{attribute 'linkalways'} 
{attribute 'no_explicit_call' := 'This FB is a CLASS and must be accessed using methods or properties'}
FUNCTION_BLOCK Feeder EXTENDS CyclicInstance IMPLEMENTS I_Feeder
VAR
	_nci : I_Nci;
	_fb : FB_NciFeedTable;
	_table : ST_NciFeedGroupTable;
	_execute : BOOL;
	_reset : BOOL;
	_feedDone : BOOL;
	_channelDone : BOOL;
	_feedBusy : BOOL;
	_resetBusy : BOOL;
	_error : BOOL;
	_errorId : UDINT;
	
	state : (IDLE, RESETTING, FEEDING, DONE, ERROR);
	command : (NONE, RESET, FEED);
	
	commandFeedback : I_CommandFeedbackReadWrite;
END_VAR

PROPERTY ChannelDone : BOOL
GET
ChannelDone := _fb.bChannelDone;
END_GET
END_PROPERTY

METHOD  CyclicCall
CASE state OF
	IDLE:
		_fb(
			bExecute := FALSE,
			bReset := FALSE,
			stNciToPlc := _nci._InternalNciPlcRef.nciToPlc,
			stFeedGroupTable := _table,
			bFeedingDone => _feedDone,
			bChannelDone => _channelDone,
			bFeedBusy => _feedBusy,
			bResetBusy => _resetBusy,
			bError => _error,
			nErrorId => _errorId
		);
		
		CASE command OF
			RESET:
				state := RESETTING;
				command := NONE;
				commandFeedback.SetBusy();
			FEED:
				state := FEEDING;
				command := NONE;
				commandFeedback.SetBusy();
		END_CASE

	RESETTING:
		_fb(
			bExecute := FALSE,
			bReset := TRUE,
			stNciToPlc := _nci._InternalNciPlcRef.nciToPlc,
			stFeedGroupTable := _table,
			bChannelDone => _channelDone,
			bFeedBusy => _feedBusy,
			bResetBusy => _resetBusy,
			bError => _error,
			nErrorId => _errorId
		);
		
		IF NOT _fb.bResetBusy THEN		
			IF _fb.bError THEN
				state := ERROR;
			ELSE
				state := DONE;
			END_IF
		END_IF

	FEEDING:
		_fb(
			bExecute := TRUE,
			bReset := FALSE,
			stNciToPlc := _nci._InternalNciPlcRef.nciToPlc,
			stFeedGroupTable := _table,
		);
		
		IF NOT _fb.bFeedBusy THEN
			IF _fb.bError THEN
				state := ERROR;
			ELSIF _fb.bFeedingDone THEN
				state := DONE;
			END_IF
		END_IF
	
	DONE:
		IF commandFeedback <> 0 THEN
			commandFeedback.SetDone();
		END_IF
		state := IDLE;		
	ERROR:
		IF commandFeedback <> 0 THEN
			commandFeedback.SetError(_fb.nErrorId);
		END_IF
		state := IDLE;
ELSE
	state := IDLE;
END_CASE
END_METHOD

METHOD FB_init : BOOL
VAR_INPUT
	bInitRetains : BOOL; // if TRUE, the retain variables are initialized (warm start / cold start)
	bInCopyCode : BOOL;  // if TRUE, the instance afterwards gets moved into the copy code (online change)
	nci : I_Nci;
END_VAR
IF nci <> 0 THEN
	_nci := nci;
END_IF
END_METHOD

METHOD FeedTable
VAR_INPUT
	table : I_Table;
	feedback : REFERENCE TO I_CommandFeedback;
END_VAR
VAR
	pCmd : POINTER TO FeederCommand;
END_VAR
IF NOT IsAlreadyExecuting() THEN
	_table := table._InternalTable;
	command := FEED;
	SetupFeedback(Feedback);
END_IF
END_METHOD

METHOD PRIVATE IsAlreadyExecuting : BOOL
IF commandFeedback = 0 THEN
	RETURN;
END_IF

IsAlreadyExecuting := commandFeedback.Busy;
END_METHOD

PROPERTY LogFeederEntries : BOOL
GET
LogFeederEntries := _fb.bLogFeederEntries;
END_GET
SET
_fb.bLogFeederEntries := LogFeederEntries;
END_SET
END_PROPERTY

METHOD Reset
VAR_INPUT
	feedback : REFERENCE TO I_CommandFeedback;
END_VAR
VAR
	pCmd : POINTER TO FeederCommand;
END_VAR
IF NOT IsAlreadyExecuting() THEN
	command := RESET;
	SetupFeedback(Feedback);
END_IF
END_METHOD

METHOD SetupFeedback : I_CommandFeedbackReadWrite
VAR_INPUT
	feedback : REFERENCE TO I_CommandFeedback;
END_VAR
VAR
	pFeedback : POINTER TO CommandFeedback;
END_VAR
IF feedback <> 0 THEN 
	feedback.Release();
END_IF

IF IsAlreadyExecuting() THEN

	IF __ISVALIDREF(feedback) THEN
		feedback := commandFeedback;
		feedback.AddReference();
	END_IF
	
	RETURN;
END_IF

IF commandFeedback <> 0 THEN 
	commandFeedback.Release();
END_IF

pFeedback := __NEW(CommandFeedback);
commandFeedback := pFeedback^;

IF __ISVALIDREF(feedback) THEN
	feedback := commandFeedback;
	feedback.AddReference();
END_IF
END_METHOD

END_FUNCTION_BLOCK

(* stored: Version 1.1.0.1, ProductVersion 3.1.4024.12
   POU Feeder: Id {9a5868fd-98f5-4278-ae73-8005b348044c}, SpecialFunc None
   Property ChannelDone: Id {ed0fa9b1-077c-4f88-8925-58f7dfbbd88b}
   Get Get: Id {3b7f5a0c-857f-4eec-9ba9-a9db8c40851f}
   Method CyclicCall: Id {de7ced26-3d49-47db-b260-0f80a2759ab5}
   Method FB_init: Id {4010d0a1-1574-46fc-a665-815377c8f205}
   Method FeedTable: Id {720b2933-f33c-4197-a656-a808090743ba}
   Method IsAlreadyExecuting: Id {138794bd-91e6-4dd8-b703-e7ba40a043b8}
   Property LogFeederEntries: Id {37494741-7336-4f81-ac4d-dd7d269806bc}
   Get Get: Id {22d7e8ef-6858-407a-b994-080d1b377908}
   Set Set: Id {ed83cacf-d3cc-4cde-86b3-578f7b21a35a}
   Method Reset: Id {79731249-b062-4e54-8eeb-562b87724ed0}
   Method SetupFeedback: Id {ad8afd8a-e417-4389-824b-d719d3e8a85d} *)
